% RSLogix 500 project flow pressure.RSS, saved by version 8.30.00.16 %
PROJECT "UNTITLED"    % processor: Bul.1763 MicroLogix 1100 Series B %

PROGRAM FILES
  LAD 2 "MAIN"  2 rungs
  LAD 3 "I/O"  12 rungs

DATA FILES
  O0 OUTPUT  4 elements
  I1 INPUT  6 elements
  S2 STATUS  66 elements
  B3 BINARY  1 elements
  T4 TIMER  1 elements
  C5 COUNTER  1 elements
  R6 CONTROL  1 elements
  N7 INTEGER  1 elements
  F8 FLOAT  1 elements

LADDER 2 "MAIN"
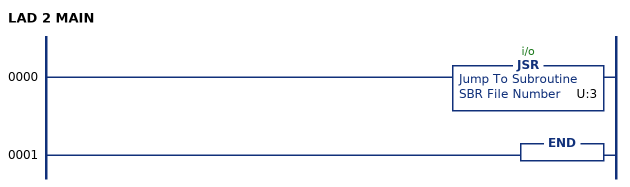
% Rung: 0 %  % edit flag set %
SOR JSR U:3 EOR
%   U:3  "i/o" %
% Rung: 1 %
SOR END EOR

LADDER 3 "I/O"
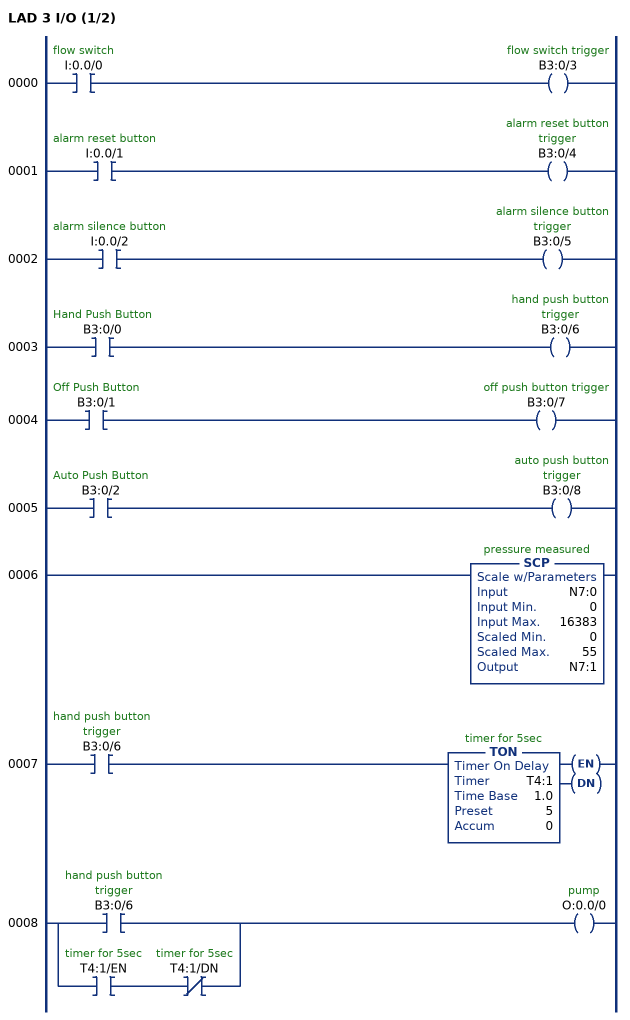
% Rung: 0 %  % edit flag set %
SOR XIC I:0.0/0 OTE B3:0/3 EOR
%   I:0.0/0  "flow switch" %
%   B3:0/3  "flow switch trigger" %
% Rung: 1 %  % edit flag set %
SOR XIC I:0.0/1 OTE B3:0/4 EOR
%   I:0.0/1  "alarm reset button" %
%   B3:0/4  "alarm reset button trigger" %
% Rung: 2 %  % edit flag set %
SOR XIC I:0.0/2 OTE B3:0/5 EOR
%   I:0.0/2  "alarm silence button" %
%   B3:0/5  "alarm silence button trigger" %
% Rung: 3 %  % edit flag set %
SOR XIC B3:0/0 OTE B3:0/6 EOR
%   B3:0/0  "Hand Push Button" %
%   B3:0/6  "hand push button trigger" %
% Rung: 4 %  % edit flag set %
SOR XIC B3:0/1 OTE B3:0/7 EOR
%   B3:0/1  "Off Push Button" %
%   B3:0/7  "off push button trigger" %
% Rung: 5 %  % edit flag set %
SOR XIC B3:0/2 OTE B3:0/8 EOR
%   B3:0/2  "Auto Push Button" %
%   B3:0/8  "auto push button trigger" %
% Rung: 6 %  % edit flag set %
SOR SCP N7:0 0 16383 0 55 N7:1 EOR
%   N7:0  "pressure sensor (0-55psi)" %
%   N7:1  "pressure measured" %
% Rung: 7 %  % edit flag set %
SOR XIC B3:0/6 TON T4:1 1.0 5 0 EOR
%   B3:0/6  "hand push button trigger" %
%   T4:1  "timer for 5sec" %
% Rung: 8 %  % edit flag set %
SOR BST XIC B3:0/6 NXB XIC T4:1/EN XIO T4:1/DN BND OTE O:0.0/0 EOR
%   B3:0/6  "hand push button trigger" %
%   T4:1  "timer for 5sec" %
%   O:0.0/0  "pump" %

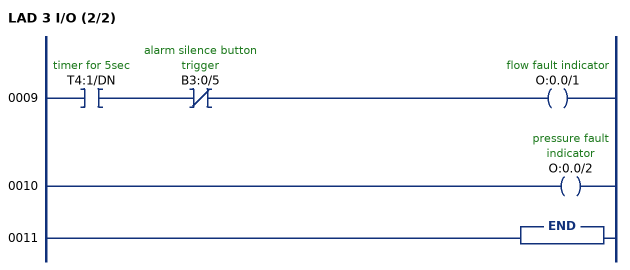
% Rung: 9 %  % edit flag set %
SOR XIC T4:1/DN XIO B3:0/5 OTE O:0.0/1 EOR
%   T4:1  "timer for 5sec" %
%   B3:0/5  "alarm silence button trigger" %
%   O:0.0/1  "flow fault indicator" %
% Rung: 10 %  % edit flag set %
SOR OTE O:0.0/2 EOR
%   O:0.0/2  "pressure fault indicator" %
% Rung: 11 %
SOR END EOR

OTHER DOCUMENTED ADDRESSES
  U:4  "controls"
